% RSLogix 500 project 10percent.RSS, saved by version 8.30.00.16 %
PROJECT "UNTITLED"    % processor: Bul.1763 MicroLogix 1100 Series A %

PROGRAM FILES
  LAD 2 "CONTINUOUS"  7 rungs
  LAD 3 "LINEAR"  9 rungs
  LAD 4 "BINARY"  9 rungs

DATA FILES
  O0 OUTPUT  4 elements
  I1 INPUT  6 elements
  S2 STATUS  66 elements
  B3 BINARY  1 elements
  T4 TIMER  1 elements
  C5 COUNTER  2 elements
  R6 CONTROL  1 elements
  N7 INTEGER  7 elements
  F8 FLOAT  1 elements
  N253 BNRYSEARCH  72 elements
  N254 LINRSEARCH  72 elements
  N255 SORTEDLIST  8 elements

LADDER 2 "CONTINUOUS"
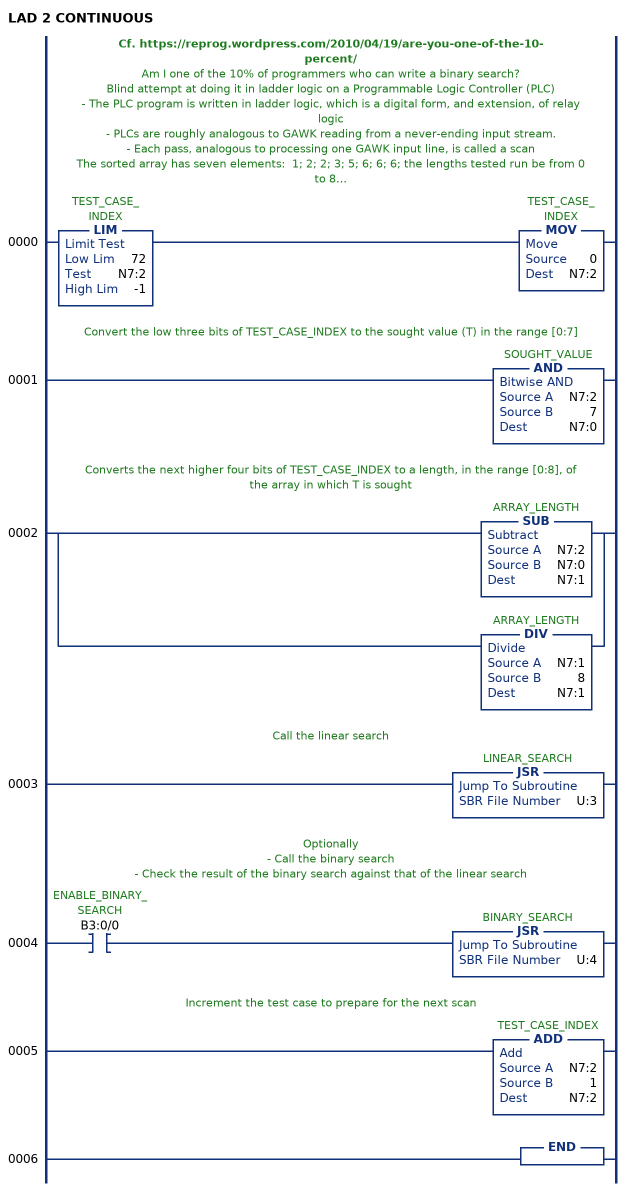
% Rung: 0 %
% TITLE: Cf. https://reprog.wordpress.com/2010/04/19/are-you-one-of-the-10-percent/ %
% Am I one of the 10% of programmers who can write a binary search?
% 
% Blind attempt at doing it in ladder logic on a Programmable Logic Controller (PLC)
% - The PLC program is written in ladder logic, which is a digital form, and extension, of relay logic
% - PLCs are roughly analogous to GAWK reading from a never-ending input stream.
%   - Each pass, analogous to processing one GAWK input line, is called a scan
% 
% The sorted array has seven elements:  1; 2; 2; 3; 5; 6; 6; 6; the lengths tested run be from 0 to 8.
% The range of sought values will be from 0 to 7.
% 
% This is the main program; on each PLC scan, this program will
% - Select one problem from the set of 72 possibilities (eight lengths and seven sought values),
% - Call the linear and binary searches
% - Compare the results %
SOR LIM 72 N7:2 -1 MOV 0 N7:2 EOR
%   N7:2  TEST_CASE_INDEX %
% Rung: 1 %
% Convert the low three bits of TEST_CASE_INDEX to the sought value (T) in the range [0:7] %
SOR AND N7:2 7 N7:0 EOR
%   N7:2  TEST_CASE_INDEX %
%   N7:0  SOUGHT_VALUE %
% Rung: 2 %
% Converts the next higher four bits of TEST_CASE_INDEX to a length, in the range [0:8], of the array in which T is sought %
SOR BST SUB N7:2 N7:0 N7:1 NXB DIV N7:1 8 N7:1 BND EOR
%   N7:2  TEST_CASE_INDEX %
%   N7:0  SOUGHT_VALUE %
%   N7:1  ARRAY_LENGTH %
% Rung: 3 %
% Call the linear search %
SOR JSR U:3 EOR
%   U:3  LINEAR_SEARCH %
% Rung: 4 %
% Optionally
% - Call the binary search
% - Check the result of the binary search against that of the linear search %
SOR XIC B3:0/0 JSR U:4 EOR
%   B3:0/0  ENABLE_BINARY_SEARCH %
%   U:4  BINARY_SEARCH %
% Rung: 5 %
% Increment the test case to prepare for the next scan %
SOR ADD N7:2 1 N7:2 EOR
%   N7:2  TEST_CASE_INDEX %
% Rung: 6 %
SOR END EOR

LADDER 3 "LINEAR"
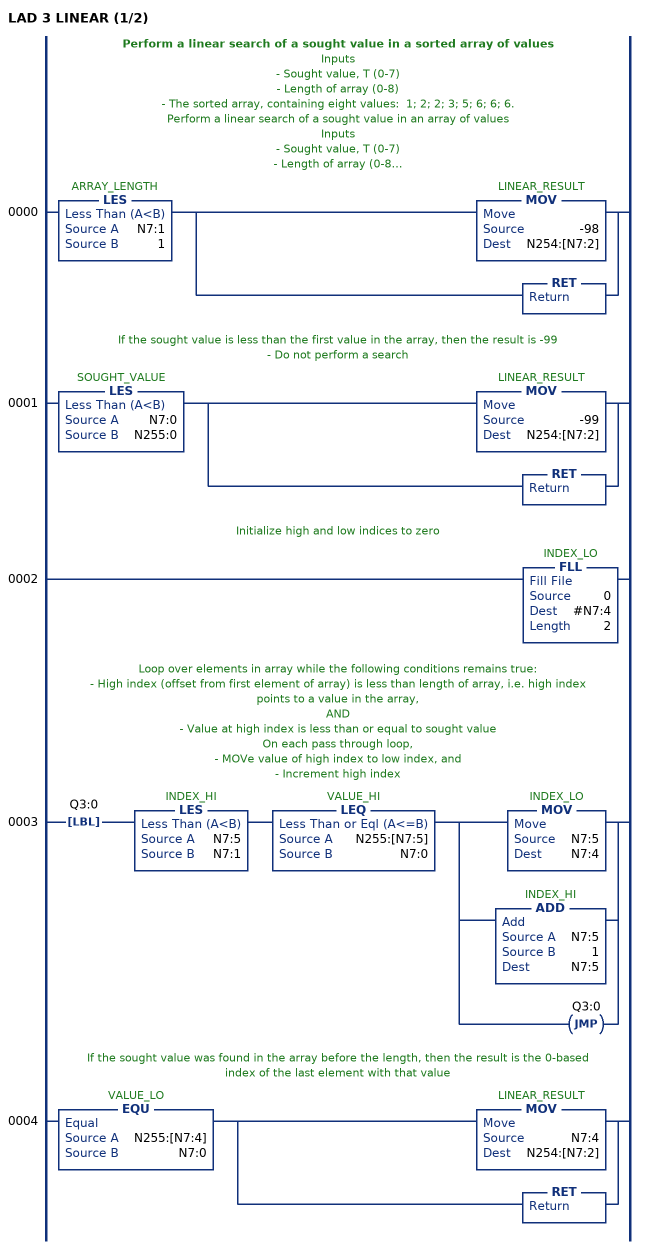
% Rung: 0 %
% TITLE: Perform a linear search of a sought value in a sorted array of values %
% Inputs
% - Sought value, T (0-7)
% - Length of array (0-8)
% - The sorted array, containing eight values:  1; 2; 2; 3; 5; 6; 6; 6.
% 
% Perform a linear search of a sought value in an array of values
% Inputs
% - Sought value, T (0-7)
% - Length of array (0-8)
% - A sorted array, containing up to eight values:  1; 2; 2; 3; 5; 6; 6; 6.
% 
% If the length of the array is less than 1, then the result is -98; don't perform a search %
SOR LES N7:1 1 BST MOV -98 N254:[N7:2] NXB RET BND EOR
%   N7:1  ARRAY_LENGTH %
%   N254:[N7:2]  LINEAR_RESULT %
%   N7:2  TEST_CASE_INDEX %
% Rung: 1 %
% If the sought value is less than the first value in the array, then the result is -99
% - Do not perform a search %
SOR LES N7:0 N255:0 BST MOV -99 N254:[N7:2] NXB RET BND EOR
%   N7:0  SOUGHT_VALUE %
%   N254:[N7:2]  LINEAR_RESULT %
%   N7:2  TEST_CASE_INDEX %
% Rung: 2 %
% Initialize high and low indices to zero %
SOR FLL 0 #N7:4 2 EOR
%   N7:4  INDEX_LO %
% Rung: 3 %
% Loop over elements in array while the following conditions remains true:
% - High index (offset from first element of array) is less than length of array, i.e. high index points to a value in the array,
% AND
% - Value at high index is less than or equal to sought value
% 
% On each pass through loop,
% - MOVe value of high index to low index, and
% - Increment high index %
SOR LBL Q3:0 LES N7:5 N7:1 LEQ N255:[N7:5] N7:0 BST MOV N7:5 N7:4 NXB ADD N7:5 1 N7:5 NXB JMP Q3:0 BND EOR
%   N7:5  INDEX_HI %
%   N7:1  ARRAY_LENGTH %
%   N255:[N7:5]  VALUE_HI %
%   N7:0  SOUGHT_VALUE %
%   N7:4  INDEX_LO %
% Rung: 4 %
% If the sought value was found in the array before the length, then the result is the 0-based index of the last element with that value %
SOR EQU N255:[N7:4] N7:0 BST MOV N7:4 N254:[N7:2] NXB RET BND EOR
%   N255:[N7:4]  VALUE_LO %
%   N7:4  INDEX_LO %
%   N7:0  SOUGHT_VALUE %
%   N254:[N7:2]  LINEAR_RESULT %
%   N7:2  TEST_CASE_INDEX %

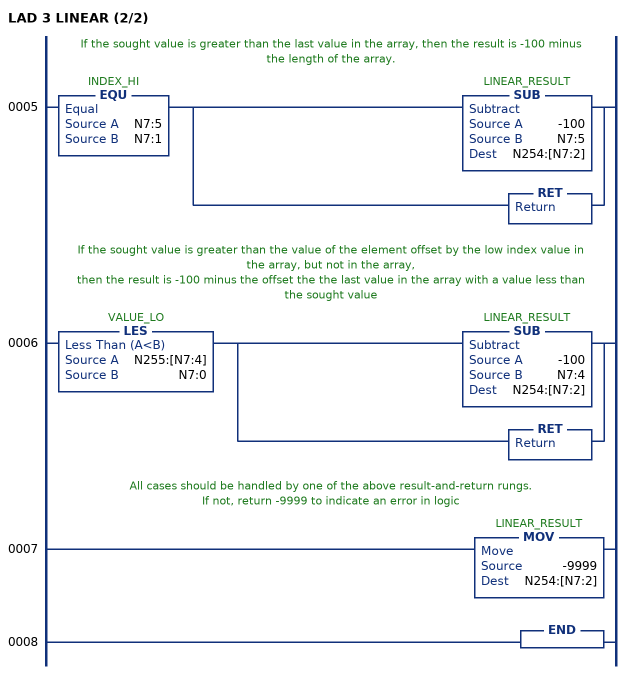
% Rung: 5 %
% If the sought value is greater than the last value in the array, then the result is -100 minus the length of the array. %
SOR EQU N7:5 N7:1 BST SUB -100 N7:5 N254:[N7:2] NXB RET BND EOR
%   N7:5  INDEX_HI %
%   N7:1  ARRAY_LENGTH %
%   N254:[N7:2]  LINEAR_RESULT %
%   N7:2  TEST_CASE_INDEX %
% Rung: 6 %
% If the sought value is greater than the value of the element offset by the low index value in the array, but not in the array,
%   then the result is -100 minus the offset the the last value in the array with a value less than the sought value %
SOR LES N255:[N7:4] N7:0 BST SUB -100 N7:4 N254:[N7:2] NXB RET BND EOR
%   N255:[N7:4]  VALUE_LO %
%   N7:4  INDEX_LO %
%   N7:0  SOUGHT_VALUE %
%   N254:[N7:2]  LINEAR_RESULT %
%   N7:2  TEST_CASE_INDEX %
% Rung: 7 %
% All cases should be handled by one of the above result-and-return rungs.
% If not, return -9999 to indicate an error in logic %
SOR MOV -9999 N254:[N7:2] EOR
%   N254:[N7:2]  LINEAR_RESULT %
%   N7:2  TEST_CASE_INDEX %
% Rung: 8 %
SOR END EOR

LADDER 4 "BINARY"
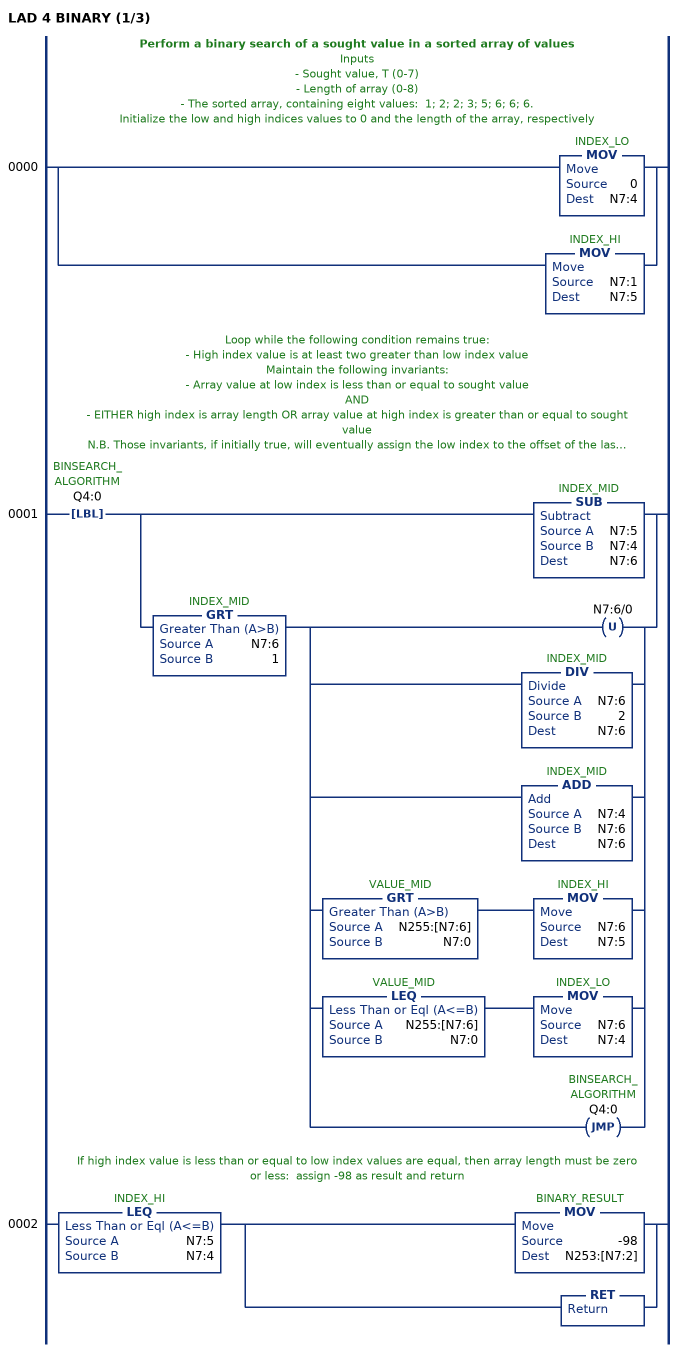
% Rung: 0 %
% TITLE: Perform a binary search of a sought value in a sorted array of values %
% Inputs
% - Sought value, T (0-7)
% - Length of array (0-8)
% - The sorted array, containing eight values:  1; 2; 2; 3; 5; 6; 6; 6.
% 
% Initialize the low and high indices values to 0 and the length of the array, respectively %
SOR BST MOV 0 N7:4 NXB MOV N7:1 N7:5 BND EOR
%   N7:4  INDEX_LO %
%   N7:1  ARRAY_LENGTH %
%   N7:5  INDEX_HI %
% Rung: 1 %
% Loop while the following condition remains true:
% - High index value is at least two greater than low index value
% 
% Maintain the following invariants:
% - Array value at low index is less than or equal to sought value
% AND
% - EITHER high index is array length OR array value at high index is greater than or equal to sought value
% 
% N.B. Those invariants, if initially true, will eventually assign the low index to the offset of the last value in the array that is less than or equal to the sought value
% N.B. Those invariants will be violated when the sought value is less than value of the first element in the array, however
%           in that case at the end the low and high index values will be 0 and 1, respectively.
% 
% On each pass through loop,
% - Calculate mid index value
% - Shift either low or high index to mid index value to maintain the invariants above %
SOR LBL Q4:0 BST SUB N7:5 N7:4 N7:6 NXB GRT N7:6 1 BST BST OTU N7:6/0 NXB DIV N7:6 2 N7:6 NXB ADD N7:4 N7:6 N7:6 BND NXB GRT N255:[N7:6] N7:0 MOV N7:6 N7:5 NXB LEQ N255:[N7:6] N7:0 MOV N7:6 N7:4 NXB JMP Q4:0 BND BND EOR
%   Q4:0  BINSEARCH_ALGORITHM %
%   N7:5  INDEX_HI %
%   N7:4  INDEX_LO %
%   N7:6  INDEX_MID %
%   N255:[N7:6]  VALUE_MID %
%   N7:0  SOUGHT_VALUE %
% Rung: 2 %
% If high index value is less than or equal to low index values are equal, then array length must be zero or less:  assign -98 as result and return %
SOR LEQ N7:5 N7:4 BST MOV -98 N253:[N7:2] NXB RET BND EOR
%   N7:5  INDEX_HI %
%   N7:4  INDEX_LO %
%   N253:[N7:2]  BINARY_RESULT %
%   N7:2  TEST_CASE_INDEX %

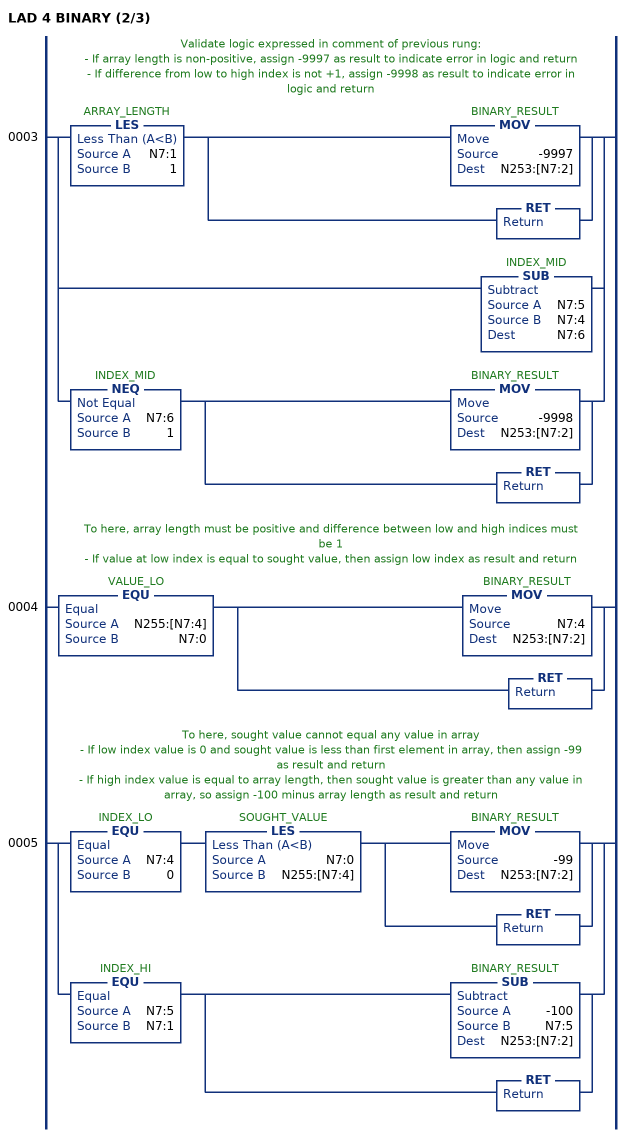
% Rung: 3 %
% Validate logic expressed in comment of previous rung:
% - If array length is non-positive, assign -9997 as result to indicate error in logic and return
% - If difference from low to high index is not +1, assign -9998 as result to indicate error in logic and return %
SOR BST LES N7:1 1 BST MOV -9997 N253:[N7:2] NXB RET BND NXB BST SUB N7:5 N7:4 N7:6 NXB NEQ N7:6 1 BST MOV -9998 N253:[N7:2] NXB RET BND BND BND EOR
%   N7:1  ARRAY_LENGTH %
%   N253:[N7:2]  BINARY_RESULT %
%   N7:2  TEST_CASE_INDEX %
%   N7:5  INDEX_HI %
%   N7:4  INDEX_LO %
%   N7:6  INDEX_MID %
% Rung: 4 %
% To here, array length must be positive and difference between low and high indices must be 1
% - If value at low index is equal to sought value, then assign low index as result and return %
SOR EQU N255:[N7:4] N7:0 BST MOV N7:4 N253:[N7:2] NXB RET BND EOR
%   N255:[N7:4]  VALUE_LO %
%   N7:4  INDEX_LO %
%   N7:0  SOUGHT_VALUE %
%   N253:[N7:2]  BINARY_RESULT %
%   N7:2  TEST_CASE_INDEX %
% Rung: 5 %
% To here, sought value cannot equal any value in array
% - If low index value is 0 and sought value is less than first element in array, then assign -99 as result and return
% - If high index value is equal to array length, then sought value is greater than any value in array, so assign -100 minus array length as result and return %
SOR BST EQU N7:4 0 LES N7:0 N255:[N7:4] BST MOV -99 N253:[N7:2] NXB RET BND NXB EQU N7:5 N7:1 BST SUB -100 N7:5 N253:[N7:2] NXB RET BND BND EOR
%   N7:4  INDEX_LO %
%   N7:0  SOUGHT_VALUE %
%   N255:[N7:4]  VALUE_LO %
%   N253:[N7:2]  BINARY_RESULT %
%   N7:2  TEST_CASE_INDEX %
%   N7:5  INDEX_HI %
%   N7:1  ARRAY_LENGTH %

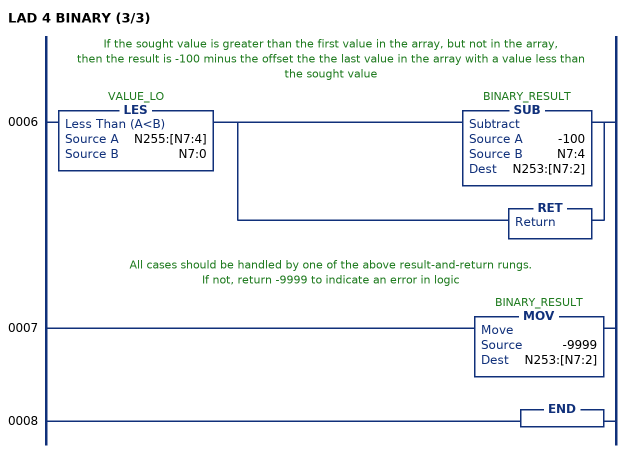
% Rung: 6 %
% If the sought value is greater than the first value in the array, but not in the array,
%   then the result is -100 minus the offset the the last value in the array with a value less than the sought value %
SOR LES N255:[N7:4] N7:0 BST SUB -100 N7:4 N253:[N7:2] NXB RET BND EOR
%   N255:[N7:4]  VALUE_LO %
%   N7:4  INDEX_LO %
%   N7:0  SOUGHT_VALUE %
%   N253:[N7:2]  BINARY_RESULT %
%   N7:2  TEST_CASE_INDEX %
% Rung: 7 %
% All cases should be handled by one of the above result-and-return rungs.
% If not, return -9999 to indicate an error in logic %
SOR MOV -9999 N253:[N7:2] EOR
%   N253:[N7:2]  BINARY_RESULT %
%   N7:2  TEST_CASE_INDEX %
% Rung: 8 %
SOR END EOR

OTHER DOCUMENTED ADDRESSES
  N7:3  ERROR_COUNT

DATA TABLE (non-zero values as saved)
DATA B3
% B3:0 % 0X0006
DATA T4
% .PRE .ACC %
% T4:0 % 1000 777
DATA C5
% .PRE .ACC %
% C5:0 % 32767 -32359
% C5:1 % 32767 24453
DATA R6
% .LEN .POS %
% R6:0 % 4 1
DATA N255
% N255:0 % 1 2 2 3 5 6 6 6
